Universal Robots PolyScope program: asm_idler_pulley_p1.urp

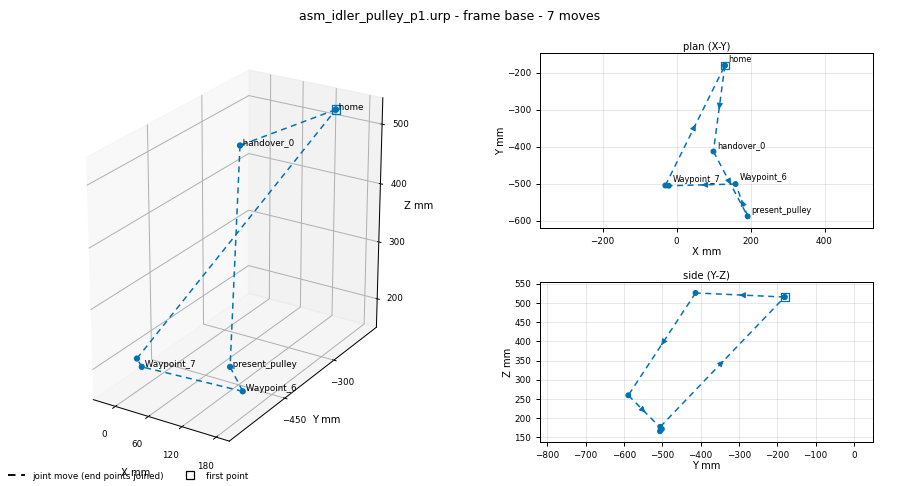
[picture p0: tool path of asm_idler_pulley_p1.urp in frame base, 7 of 8 moves have a stored position in this frame; points joined in program order, loops and branches not executed]
Program asm_idler_pulley_p1 (installation=default directory=/programs/wrs2020 createdIn=3.8.0.61336 lastSavedIn=5.10.0.106288 robotSerialNumber=20205500607)
Calibrated DH parameters: a=[0.000096, -0.337, -0.383372, 0.000118, 0.000015, 0]; d=[0.162724, 79.377998, -95.545185, 16.300583, 0.099689, 0.099499]; alpha=[1.569249, 0.003272, 0.005201, 1.570041, -1.570219, 0]; deltaTheta=[0, 0.65664, 5.410619, 0.215927, -0.000001, 0]
Robot Program (runOnlyOnce=true)
  MoveJ speed 60 deg/s, acceleration 80 deg/s^2 (useActiveTCP=false) tcp=gripper_85_tip; feature=Base
    currentpose := get_actual_joint_positions()
    Waypoint Waypoint (Variable): variable=currentpose
    Waypoint home: TCP in base x=130.657 y=-180.679 z=515.923 mm, rx=-0.0119 ry=-3.1403 rz=-0.0318 rad; joints [89.953, -120.322, 80.217, -48.701, -89.954, 0.005] deg; TCP offset x=0 y=0 z=165 mm, rx=0 ry=0 rz=0 rad
    Popup Message (haltProgram=false message=wait for a_bot to hold pin, Continue to pick it inputType=Text)
    URCap Gripper (Robotiq_Grippers, Robotiq Inc.) dataModel(position=100.0, force=100.0, speed=100.0, positionInDouble=100.0, forceInDouble=100.0, speedInDouble=100.0, slaveIds=[9], blocking=false)
    Waypoint handover_0: TCP in base x=99.663 y=-413.108 z=526.627 mm, rx=0.0095 ry=2.2256 rz=-2.2108 rad; joints [76.279, -128.98, 138.408, -189.062, -76.136, 0.581] deg
    SuppressedNode
      Waypoint looking_at_belt: TCP in base x=162.548 y=-458.764 z=158.73 mm, rx=-1.6745 ry=-2.0805 rz=0.6897 rad; joints [112.15, -80.245, 110.523, -113.873, -125.384, 101.857] deg
  Folder Touch+Grasp
    MoveL speed 250 mm/s, acceleration 1200 mm/s^2 (useActiveTCP=true) feature=Base
      MoveDirectionNode (selectedDirection=ZPlus toolParams=0.01, 0.05) feature=Base
        Until TOOL_CONTACT_DETECTION (allowActions=false retraction=0 decelerationAcceleration=3 decelerationAngularAcceleration=34.906585)
    URCap Gripper (Robotiq_Grippers, Robotiq Inc.) dataModel(position=60.3921568627451, force=100.0, speed=100.0, positionInDouble=60.3921568627451, forceInDouble=100.0, speedInDouble=100.0, slaveIds=[9], blocking=true)
    MoveL speed 250 mm/s, acceleration 1200 mm/s^2 (useActiveTCP=true) feature=Base
      MoveDirectionNode (selectedDirection=ZPlus)
        Until DISTANCE (allowActions=false deceleration=3 distanceNodeType=STOP) Distance=0.009; motionParameters(blendRadius=0)
    URCap Gripper (Robotiq_Grippers, Robotiq Inc.) dataModel(position=100.0, force=100.0, speed=100.0, positionInDouble=100.0, forceInDouble=100.0, speedInDouble=100.0, slaveIds=[9], blocking=false)
  Popup Message (haltProgram=false message=wait for a_bot to release, Continue to move down inputType=Text)
  MoveJ speed 60 deg/s, acceleration 80 deg/s^2 (useActiveTCP=true) feature=Base
    Waypoint present_pulley: TCP in base x=192.248 y=-588.457 z=259.678 mm, rx=0.0094 ry=2.2258 rz=-2.2107 rad; joints [100.087, -59.68, 129.181, -249.019, -100.325, 0.794] deg
  Popup Message (haltProgram=false message=wait for a_bot to stack 3 parts. Continue to move into ridge inputType=Text)
  MoveJ speed 60 deg/s, acceleration 120 deg/s^2 (useActiveTCP=false) tcp=gripper_85_tip; feature=Base
    Waypoint Waypoint_6: TCP in base x=159.447 y=-501.036 z=171.589 mm, rx=2.0868 ry=1.9752 rz=-0.8061 rad; joints [104.097, -87.703, 124.272, -151.013, -111.848, 102.545] deg
    Waypoint Waypoint_7: TCP in base x=-21.054 y=-505.778 z=166.036 mm, rx=1.9773 ry=2.0556 rz=-0.7883 rad; joints [75.454, -94.313, 133.938, -161.728, -95.327, 71.8] deg
    Waypoint Waypoint_8: TCP in base x=-30.311 y=-505.122 z=177.558 mm, rx=1.9536 ry=1.9163 rz=-0.5046 rad; joints [65.052, -98.219, 132.305, -151.087, -78.086, 69.08] deg
  SuppressedNode
    MoveL speed 20 mm/s, acceleration 50 mm/s^2 (useActiveTCP=true) feature=Base
      MoveDirectionNode (selectedDirection=XMinus)
        Until TOOL_CONTACT_DETECTION (allowActions=false retraction=0 decelerationAcceleration=3 decelerationAngularAcceleration=34.906585)
  Popup Message (haltProgram=false message=wait for abot to take stack. c to release and get tool inputType=Text)
  URCap Gripper (Robotiq_Grippers, Robotiq Inc.) dataModel(position=58.431372549019606, force=100.0, speed=100.0, positionInDouble=58.431372549019606, forceInDouble=100.0, speedInDouble=100.0, slaveIds=[9], blocking=true)
  MoveL speed 250 mm/s, acceleration 1200 mm/s^2 (useActiveTCP=true) feature=Base
    MoveDirectionNode (selectedDirection=XPlus)
      Until DISTANCE (allowActions=false deceleration=3 distanceNodeType=STOP) Distance=0.1; motionParameters(blendRadius=0)
  MoveJ speed 60 deg/s, acceleration 80 deg/s^2 (useActiveTCP=true) feature=Base
    Waypoint home: TCP in base x=130.657 y=-180.679 z=515.923 mm, rx=-0.0119 ry=-3.1403 rz=-0.0318 rad; joints [89.953, -120.322, 80.217, -48.701, -89.954, 0.005] deg
  SuppressedNode
    Popup Message (haltProgram=false message=take padless tool, go to horizontal ready. c to move with tool inputType=Text)
  'next: p2'
